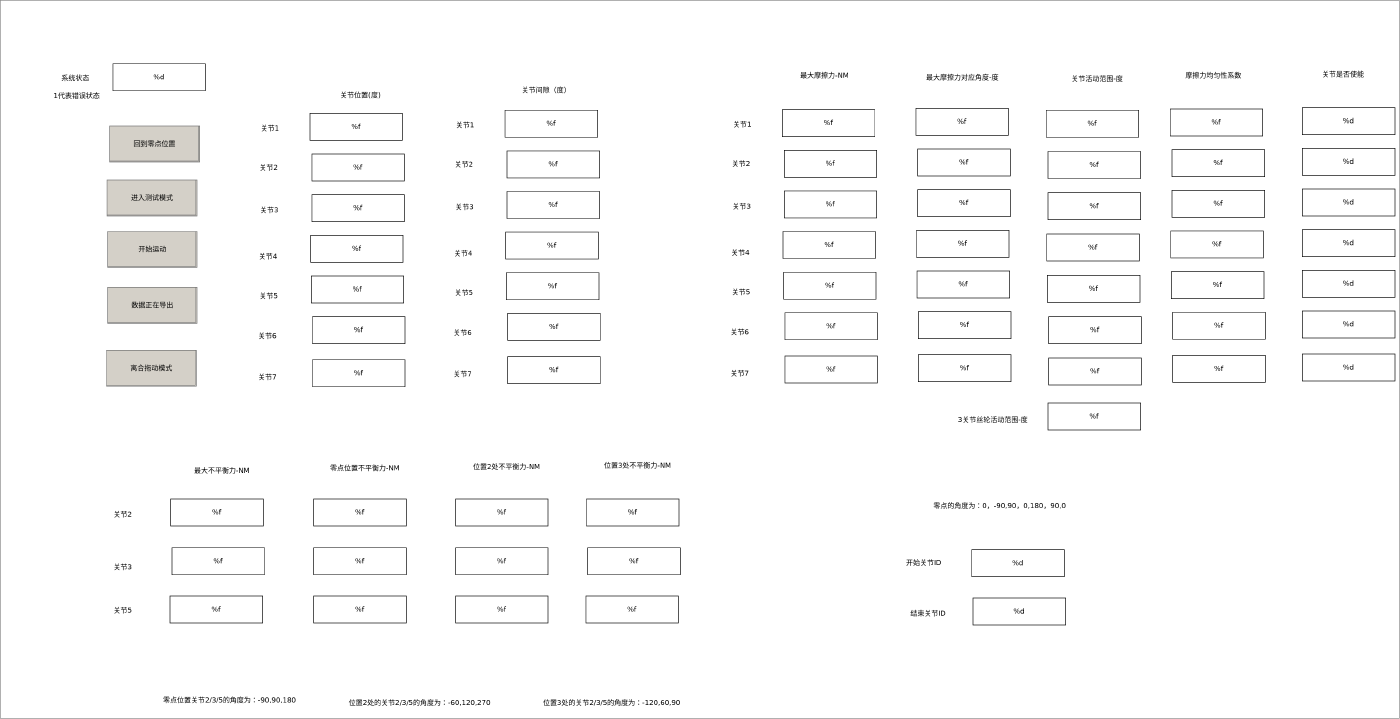
VISUALIZATION friction_a2  // 2202x1132
    Button (168,283 142x57), "进入测试模式", colour toggle: g_frictionTest.m_testMode[2]
        toggle g_frictionTest.m_testMode[2]
    Button (169,364 141x57), "开始运动", colour toggle: g_frictionTest.m_startMotion[2]
        toggle g_frictionTest.m_startMotion[2]
    Rectangle (487,178 146x43), "%f", text variable: g_frictionTest.m_armDHJntPos[2][1]
    Label (373,184 103x36), "关节1"
    Label (371,246 103x36), "关节2"
    Label (372,313 103x36), "关节3"
    Label (370,386 103x36), "关节4"
    Label (371,448 103x36), "关节5"
    Label (369,511 103x36), "关节6"
    Label (369,576 103x36), "关节7"
    Rectangle (490,242 146x43), "%f", text variable: g_frictionTest.m_armDHJntPos[2][2]
    Rectangle (490,306 146x43), "%f", text variable: g_frictionTest.m_armDHJntPos[2][3]
    Rectangle (488,370 146x43), "%f", text variable: g_frictionTest.m_armDHJntPos[2][4]
    Rectangle (489,434 146x43), "%f", text variable: g_frictionTest.m_armDHJntPos[2][5]
    Rectangle (491,498 146x43), "%f", text variable: g_frictionTest.m_armDHJntPos[2][6]
    Rectangle (491,566 146x43), "%f", text variable: g_frictionTest.m_armDHJntPos[2][7]
    Button (167,551 142x57), "离合拖动模式", colour toggle: g_frictionTest.m_clutchMode[2]
        toggle g_frictionTest.m_clutchMode[2]
    Rectangle (794,173 146x43), "%f", text variable: g_frictionTest.m_jntGap[2][1]
    Label (680,179 103x36), "关节1"
    Label (678,241 103x36), "关节2"
    Label (679,308 103x36), "关节3"
    Label (677,381 103x36), "关节4"
    Label (678,443 103x36), "关节5"
    Label (676,506 103x36), "关节6"
    Label (676,571 103x36), "关节7"
    Rectangle (797,237 146x43), "%f", text variable: g_frictionTest.m_jntGap[2][2]
    Rectangle (797,301 146x43), "%f", text variable: g_frictionTest.m_jntGap[2][3]
    Rectangle (795,365 146x43), "%f", text variable: g_frictionTest.m_jntGap[2][4]
    Rectangle (796,429 146x43), "%f", text variable: g_frictionTest.m_jntGap[2][5]
    Rectangle (798,493 146x43), "%f", text variable: g_frictionTest.m_jntGap[2][6]
    Rectangle (798,561 146x43), "%f", text variable: g_frictionTest.m_jntGap[2][7]
    Label (118,795 150x30), "关节2"
    Label (118,878 150x30), "关节3"
    Label (118,946 150x30), "关节5"
    Rectangle (268,785 146x43), "%f", text variable: g_frictionTest.m_unbalancedMax[2][2]
    Label (274,726 150x30), "最大不平衡力-NM"
    Rectangle (270,862 146x43), "%f", text variable: g_frictionTest.m_unbalancedMax[2][3]
    Rectangle (267,938 146x43), "%f", text variable: g_frictionTest.m_unbalancedMax[2][5]
    Rectangle (493,785 146x43), "%f", text variable: g_frictionTest.m_jntTestPntUnbalancedTrq[2,2,1]
    Label (499,722 150x30), "零点位置不平衡力-NM"
    Rectangle (493,862 146x43), "%f", text variable: g_frictionTest.m_jntTestPntUnbalancedTrq[2,3,1]
    Rectangle (493,938 146x43), "%f", text variable: g_frictionTest.m_jntTestPntUnbalancedTrq[2,5,1]
    Rectangle (716,785 146x43), "%f", text variable: g_frictionTest.m_jntTestPntUnbalancedTrq[2,2,2]
    Label (722,720 150x30), "位置2处不平衡力-NM"
    Rectangle (716,862 146x43), "%f", text variable: g_frictionTest.m_jntTestPntUnbalancedTrq[2,3,2]
    Rectangle (716,938 146x43), "%f", text variable: g_frictionTest.m_jntTestPntUnbalancedTrq[2,5,2]
    Rectangle (922,785 146x43), "%f", text variable: g_frictionTest.m_jntTestPntUnbalancedTrq[2,2,3]
    Label (928,718 150x30), "位置3处不平衡力-NM"
    Rectangle (924,862 146x43), "%f", text variable: g_frictionTest.m_jntTestPntUnbalancedTrq[2,3,3]
    Rectangle (921,938 146x43), "%f", text variable: g_frictionTest.m_jntTestPntUnbalancedTrq[2,5,3]
    Button (169,452 141x57), "数据正在导出", colour toggle: g_frictionTest.m_duringWriteData[2]
    Label (210,1077 302x51), "零点位置关节2/3/5的角度为：-90,90,180"
    Label (509,1081 302x51), "位置2处的关节2/3/5的角度为：-60,120,270"
    Label (811,1081 302x51), "位置3处的关节2/3/5的角度为：-120,60,90"
    Label (1378,871 150x30), "开始关节ID"
    Rectangle (1528,865 146x43), "%d", text variable: g_frictionTest.m_jntIdStart[2]
        OnMouseClick: write the text variable via Default
    Label (1385,951 150x30), "结束关节ID"
    Rectangle (1530,941 146x43), "%d", text variable: g_frictionTest.m_jntIdEnd[2]
        OnMouseClick: write the text variable via Default
    Label (1405,770 335x53), "零点的角度为：0，-90,90，0,180，90,0"
    Label (492,135 150x30), "关节位置(度)"
    Label (784,127 150x30), "关节间隙（度）"
    Rectangle (1230,172 146x43), "%f", text variable: g_frictionTest.m_CoulombFrictionMax[2][1]
    Label (1116,178 103x36), "关节1"
    Label (1114,240 103x36), "关节2"
    Label (1115,307 103x36), "关节3"
    Label (1113,380 103x36), "关节4"
    Label (1114,442 103x36), "关节5"
    Label (1112,505 103x36), "关节6"
    Label (1112,570 103x36), "关节7"
    Rectangle (1233,236 146x43), "%f", text variable: g_frictionTest.m_CoulombFrictionMax[2][2]
    Rectangle (1233,300 146x43), "%f", text variable: g_frictionTest.m_CoulombFrictionMax[2][3]
    Rectangle (1231,364 146x43), "%f", text variable: g_frictionTest.m_CoulombFrictionMax[2][4]
    Rectangle (1232,428 146x43), "%f", text variable: g_frictionTest.m_CoulombFrictionMax[2][5]
    Rectangle (1234,492 146x43), "%f", text variable: g_frictionTest.m_CoulombFrictionMax[2][6]
    Rectangle (1234,560 146x43), "%f", text variable: g_frictionTest.m_CoulombFrictionMax[2][7]
    Label (1222,104 150x30), "最大摩擦力-NM"
    Rectangle (1440,170 146x43), "%f", text variable: g_frictionTest.m_CoulombFrictionMax_JntPos[2][1]
    Rectangle (1443,234 146x43), "%f", text variable: g_frictionTest.m_CoulombFrictionMax_JntPos[2][2]
    Rectangle (1443,298 146x43), "%f", text variable: g_frictionTest.m_CoulombFrictionMax_JntPos[2][3]
    Rectangle (1441,362 146x43), "%f", text variable: g_frictionTest.m_CoulombFrictionMax_JntPos[2][4]
    Rectangle (1442,426 146x43), "%f", text variable: g_frictionTest.m_CoulombFrictionMax_JntPos[2][5]
    Rectangle (1444,490 146x43), "%f", text variable: g_frictionTest.m_CoulombFrictionMax_JntPos[2][6]
    Rectangle (1444,558 146x43), "%f", text variable: g_frictionTest.m_CoulombFrictionMax_JntPos[2][7]
    Label (1397,107 233x30), "最大摩擦力对应角度-度"
    Rectangle (1645,173 146x43), "%f", text variable: g_frictionTest.m_jntMotRange[2][1]
    Rectangle (1648,238 146x43), "%f", text variable: g_frictionTest.m_jntMotRange[2][2]
    Rectangle (1648,303 146x43), "%f", text variable: g_frictionTest.m_jntMotRange[2][3]
    Rectangle (1646,368 146x43), "%f", text variable: g_frictionTest.m_jntMotRange[2][4]
    Rectangle (1647,433 146x43), "%f", text variable: g_frictionTest.m_jntMotRange[2][5]
    Rectangle (1649,498 146x43), "%f", text variable: g_frictionTest.m_jntMotRange[2][6]
    Rectangle (1649,563 146x43), "%f", text variable: g_frictionTest.m_jntMotRange[2][7]
    Label (1609,109 233x30), "关节活动范围-度"
    Button (172,198 142x57), "回到零点位置", colour toggle: g_frictionTest.m_getHome[2]
        tap g_frictionTest.m_getHome[2]
    Rectangle (177,100 146x43), "%d", text variable: g_systemInfo.m_masterArmState[2]
    Label (67,105 103x36), "系统状态"
    Label (69,133 103x36), "1代表错误状态"
    Rectangle (1648,634 146x43), "%f", text variable: g_frictionTest.m_jntMotRangeJ3[2]
    Label (1496,646 131x30), "3关节丝轮活动范围-度"
    Rectangle (1840,171 146x43), "%f", text variable: g_frictionTest.m_CoulombFrictionRatio[2,1]
    Rectangle (1843,235 146x43), "%f", text variable: g_frictionTest.m_CoulombFrictionRatio[2,2]
    Rectangle (1843,299 146x43), "%f", text variable: g_frictionTest.m_CoulombFrictionRatio[2,3]
    Rectangle (1841,363 146x43), "%f", text variable: g_frictionTest.m_CoulombFrictionRatio[2,4]
    Rectangle (1842,427 146x43), "%f", text variable: g_frictionTest.m_CoulombFrictionRatio[2,5]
    Rectangle (1844,491 146x43), "%f", text variable: g_frictionTest.m_CoulombFrictionRatio[2,6]
    Rectangle (1844,559 146x43), "%f", text variable: g_frictionTest.m_CoulombFrictionRatio[2,7]
    Label (1819,104 179x30), "摩擦力均匀性系数"
    Rectangle (2048,169 146x43), "%d", text variable: g_frictionTest.m_jntEnable[2,1]
        OnMouseClick: write the text variable via Default
    Label (2023,102 179x30), "关节是否使能"
    Rectangle (2048,233 146x43), "%d", text variable: g_frictionTest.m_jntEnable[2,2]
        OnMouseClick: write the text variable via Default
    Rectangle (2048,297 146x43), "%d", text variable: g_frictionTest.m_jntEnable[2,3]
        OnMouseClick: write the text variable via Default
    Rectangle (2048,361 146x43), "%d", text variable: g_frictionTest.m_jntEnable[2,4]
        OnMouseClick: write the text variable via Default
    Rectangle (2048,425 146x43), "%d", text variable: g_frictionTest.m_jntEnable[2,5]
        OnMouseClick: write the text variable via Default
    Rectangle (2048,489 146x43), "%d", text variable: g_frictionTest.m_jntEnable[2,6]
        OnMouseClick: write the text variable via Default
    Rectangle (2048,557 146x43), "%d", text variable: g_frictionTest.m_jntEnable[2,7]
        OnMouseClick: write the text variable via Default
END_VISUALIZATION

(* stored: Version 1.1.0.1, ProductVersion 3.1.4024.11
   Visu friction_a2: Id {f383995d-5ad3-4add-837a-3b43b8dc352b} *)
